// TIA Portal V19 export
DATA_BLOCK "DI_FW_Auftrag_DB"   // DB9
// stored: AutoNumber false, InstanceOfName FB_FW_Auftrag, InstanceOfType FB
"FB_FW_Auftrag"
   // VAR
   //    StepNbr : Int;
   //    Quelle : Int;
   //    Ziel : Int;
   //    Positionen { S7_SetPoint := 'True'} : Array[1..30] of "UDT_Auftrag_Pos";
   //    Frg_Einfahrt { S7_SetPoint := 'True'} : Bool;
   //    Frg_Ausfahrt : Bool;
   //    Frg_Ablauf : Bool;
   // END_VAR
BEGIN
END_DATA_BLOCK
